// TIA Portal project "Grundkurs Aufgabe 8 NEU" (V15.1)
// Vorlageprojekt für das Buch mit Zielsystem S7-1200

(* hardware
DEVICE "S7-1200-Station_1"  S7-1200 Station
   slot 0: "Baugruppenträger_0"  Rack  V1.0
   slot 1: "SPS"  CPU 1212C AC/DC/Rly  6ES7 212-1BE40-0XB0  V4.2
*)

// ===== PLC "SPS"  CPU 1212C AC/DC/Rly =====

VAR_GLOBAL   // PLC tag table "Eingänge und Ausgänge"
   "Taster_Ebene1" AT %E0.0 : Bool;   // Taster Bedienpult Ebene 1 anfahren (Schließer)
   "Taster_Ebene2" AT %E0.1 : Bool;   // Taster Bedienpult Ebene 2 anfahren (Schließer)
   "Taster_Ebene3" AT %E0.2 : Bool;   // Taster Bedienpult Ebene 3 anfahren (Schließer)
   "Sensor_Ebene1" AT %E0.3 : Bool;   // Sensor Aufzug Ebene 1 erreicht (Schließer)
   "Sensor_Ebene2" AT %E0.4 : Bool;   // Sensor Aufzug Ebene 2 erreicht (Schließer)
   "Sensor_Ebene3" AT %E0.5 : Bool;   // Sensor Aufzug Ebene 3 erreicht (Schließer)
   "Leuchte_Ebene1" AT %A0.0 : Bool;   // Leuchte Bedienpult Ebene 1 erreicht
   "Leuchte_Ebene2" AT %A0.1 : Bool;   // Leuchte Bedienpult Ebene 2 erreicht
   "Leuchte_Ebene3" AT %A0.2 : Bool;   // Leuchte Bedienpult Ebene 3 erreicht
   "Motor_Aufzug_heben" AT %A0.3 : Bool;   // Aufzug nach oben fahren
   "Motor_Aufzug_senken" AT %A0.4 : Bool;   // Aufzug nach unten fahren
END_VAR

VAR_GLOBAL   // PLC tag table "Merker"
   "Ebene1_anfahren" AT %M1.0 : Bool;   // Aufzug auf Ebene 1 fahren
   "Ebene2_anfahren" AT %M1.1 : Bool;   // Aufzug auf Ebene 2 fahren
   "Ebene3_anfahren" AT %M1.2 : Bool;   // Aufzug auf Ebene 3 fahren
   "Aufzug_heben" AT %M2.0 : Bool;   // Aufzug nach oben fahren
   "Aufzug_senken" AT %M2.1 : Bool;   // Aufzug nach unten fahren
END_VAR

FUNCTION "Kopplung_FactoryIO_mit_PLCSIM" : Void   // FC9000, SCL
{ S7_Optimized_Access := 'TRUE' }
VERSION : 0.1
   VAR_TEMP
      rdTimeReturn : Int;
      outputTime : DTL;
      SyncVal : Byte;
      forVal : Int;
      forVal_2 : Int;
      Value : Byte;
   END_VAR
   VAR CONSTANT
      CompVal : Byte := 16#34;
      Value_01 : Byte := 16#11;
      Value_01_DW : DWord := 16#A165_D992;
      Value_02_DW : DWord := 16#58BE_4401;
   END_VAR
BEGIN

   #Value:=PEEK(area := 16#82,
        dbNumber := 0,
        byteOffset := 511);
   #Value := #Value + 1;

   POKE(area := 16#82,
        dbNumber := 0,
        byteOffset := 511,
        value := #Value);

   POKE(area:=16#81,
        dbNumber:=0,
        byteOffset:=1016,
        value:=#Value_01_DW);
   POKE(area := 16#81,
        dbNumber := 0,
        byteOffset := 1020,
        value := #Value_02_DW);

   POKE(area := 16#81,
        dbNumber := 0,
        byteOffset := 511,
        value := B#16#00);

   FOR #forVal := 0 TO 120 DO
       FOR #forVal_2:=0 TO 10 DO
           #rdTimeReturn:=RD_SYS_T(#outputTime);
           #rdTimeReturn := WR_SYS_T(#outputTime);
           #rdTimeReturn := RD_SYS_T(#outputTime);
           #rdTimeReturn := WR_SYS_T(#outputTime);
       END_FOR;
       #SyncVal:= PEEK(area := 16#81,
                      dbNumber := 0,
                      byteOffset := 511);
       IF #SyncVal = #CompVal THEN
          GOTO M_1;
       END_IF;
   END_FOR;
   RETURN;

   M_1:
   POKE(area := 16#81,
        dbNumber := 0,
        byteOffset := 511,
        value := B#16#0);
END_FUNCTION

ORGANIZATION_BLOCK "Main"   // OB1, FBD, ProgramCycle
TITLE = "Main Program Sweep (Cycle)"
{ S7_Optimized_Access := 'TRUE' }
VERSION : 0.1
   VAR_INPUT
      Initial_Call : Bool;   // Initial call of this OB
      Remanence : Bool;   // =True, if remanent data are available
   END_VAR
BEGIN

REGION Network 1: Konnektierungsbaustein für PLC-Lab / Bausteinaufruf FC9000 (Für Aufgabe nicht relevant)
   // Im Netzwerk 1 wird der Konnektierungsbaustein für PLC-Lab aufgerufen.
   // Dieser Aufruf darf nicht entfernt werden!
   // Der Baustein FC9000 organisiert den Datentransfer zwischen PLCSIM und FactoryIO.
   // Der Baustein kann als Beispielprojekt von der FactoryIO-Homepage heruntergeladen werden.
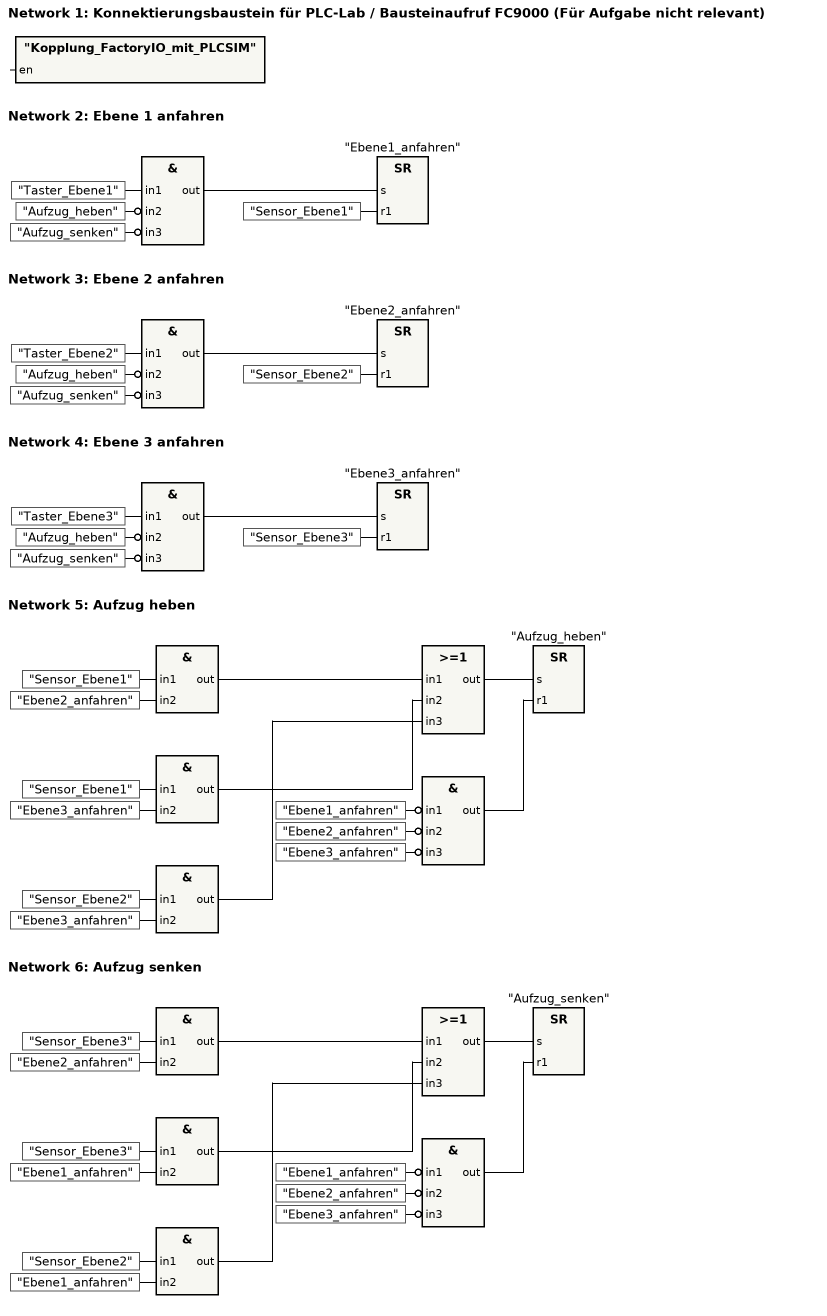
   "Kopplung_FactoryIO_mit_PLCSIM"();
END_REGION

REGION Network 2: Ebene 1 anfahren
   IF "Taster_Ebene1" AND NOT "Aufzug_heben" AND NOT "Aufzug_senken" THEN
       "Ebene1_anfahren" := TRUE;   // SR flip-flop
   END_IF;
   IF "Sensor_Ebene1" THEN "Ebene1_anfahren" := FALSE; END_IF;
END_REGION

REGION Network 3: Ebene 2 anfahren
   IF "Taster_Ebene2" AND NOT "Aufzug_heben" AND NOT "Aufzug_senken" THEN
       "Ebene2_anfahren" := TRUE;   // SR flip-flop
   END_IF;
   IF "Sensor_Ebene2" THEN "Ebene2_anfahren" := FALSE; END_IF;
END_REGION

REGION Network 4: Ebene 3 anfahren
   IF "Taster_Ebene3" AND NOT "Aufzug_heben" AND NOT "Aufzug_senken" THEN
       "Ebene3_anfahren" := TRUE;   // SR flip-flop
   END_IF;
   IF "Sensor_Ebene3" THEN "Ebene3_anfahren" := FALSE; END_IF;
END_REGION

REGION Network 5: Aufzug heben
   IF ("Sensor_Ebene1" AND "Ebene2_anfahren") OR ("Sensor_Ebene1" AND "Ebene3_anfahren") OR ("Sensor_Ebene2" AND "Ebene3_anfahren") THEN
       "Aufzug_heben" := TRUE;   // SR flip-flop
   END_IF;
   IF NOT "Ebene1_anfahren" AND NOT "Ebene2_anfahren" AND NOT "Ebene3_anfahren" THEN
       "Aufzug_heben" := FALSE;
   END_IF;
END_REGION

REGION Network 6: Aufzug senken
   IF ("Sensor_Ebene3" AND "Ebene2_anfahren") OR ("Sensor_Ebene3" AND "Ebene1_anfahren") OR ("Sensor_Ebene2" AND "Ebene1_anfahren") THEN
       "Aufzug_senken" := TRUE;   // SR flip-flop
   END_IF;
   IF NOT "Ebene1_anfahren" AND NOT "Ebene2_anfahren" AND NOT "Ebene3_anfahren" THEN
       "Aufzug_senken" := FALSE;
   END_IF;
END_REGION

REGION Network 7: Leuchte Bedienpult Ebene 1 erreicht
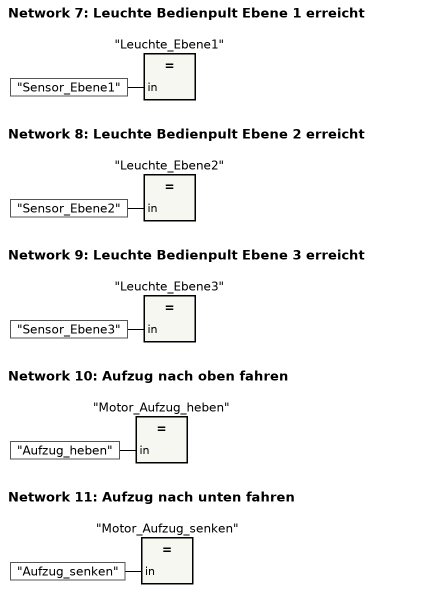
   "Leuchte_Ebene1" := "Sensor_Ebene1";
END_REGION

REGION Network 8: Leuchte Bedienpult Ebene 2 erreicht
   "Leuchte_Ebene2" := "Sensor_Ebene2";
END_REGION

REGION Network 9: Leuchte Bedienpult Ebene 3 erreicht
   "Leuchte_Ebene3" := "Sensor_Ebene3";
END_REGION

REGION Network 10: Aufzug nach oben fahren
   "Motor_Aufzug_heben" := "Aufzug_heben";
END_REGION

REGION Network 11: Aufzug nach unten fahren
   "Motor_Aufzug_senken" := "Aufzug_senken";
END_REGION
END_ORGANIZATION_BLOCK